(* IEC 61131-3 sources: CODESYS-IO-Visualization/CODESYS-IO-Visualization.fbsproj/Subs/Instruments, 10 files *)

(* ---- Accum.prg.st ---- *)
PROGRAM Accum

VAR_IN_OUT
	Data: Accum_UDT;
END_VAR

VAR
END_VAR

CycleTime(value := Data.CT);
Data.SampleSeconds := Data.SampleSeconds + Data.CT.Sec;

IF (NOT Data.Enable) THEN
	Data.LastEnable := FALSE;
	RETURN;
END_IF;

IF (Data.ValueIn_Realtime < Data.ZeroLimit) THEN
	Data.ValueIn_Realtime := 0.0;
END_IF;

// Set Min / Max Values
IF (Data.ValueIn_Realtime < Data.Value[0].ValueMin) THEN
	Data.Value[0].ValueMin := Data.ValueIn_Realtime;
END_IF;

IF (Data.ValueIn_Realtime > Data.Value[0].ValueMax) THEN
	Data.Value[0].ValueMax := Data.ValueIn_Realtime;
END_IF;

// Check to see if it's time to reset the Total
CASE Data.Period OF
	0: // Manual Reset
		Data.ResetInProcess := Data.Reset OR Data.ResetInternal;
	1: // Hourly
		Data.ResetInProcess := (((Lib_GVL.ClockLocal.Minute = Data.RollMinute) AND (Lib_GVL.ClockLocal.Second < 5)) OR Data.Reset);
	2: // Daily
		Data.ResetInProcess := (((Lib_GVL.ClockLocal.Hour = Data.RollHour) AND (Lib_GVL.ClockLocal.Minute = Data.RollMinute) AND (Lib_GVL.ClockLocal.Second < 5)) OR Data.Reset);
	3: // Monthly
		Data.ResetInProcess := (((Lib_GVL.ClockLocal.Day = Data.RollDay) AND (Lib_GVL.ClockLocal.Hour = Data.RollHour) AND (Lib_GVL.ClockLocal.Minute = Data.RollMinute) AND (Lib_GVL.ClockLocal.Second < 5)) OR Data.Reset);
	4: // Yearly
		Data.ResetInProcess := (((Lib_GVL.ClockLocal.Month = Data.RollMonth) AND (Lib_GVL.ClockLocal.Day = Data.RollDay) AND (Lib_GVL.ClockLocal.Hour = Data.RollHour) AND (Lib_GVL.ClockLocal.Minute = Data.RollMinute) AND (Lib_GVL.ClockLocal.Second < 5)) OR Data.Reset);
END_CASE;

Data.ResetAccumulator := Data.ResetInProcess;

IF (Data.ResetInProcess) THEN	// Always Accum if we are about to reset.
	Data.DoAccum := (Data.SampleSeconds > 0.0);
ELSE  // Only totalize so oftem to limit math errors.  If time change is too big, don't accum this likely means the system clock was updated, just skip it.
	IF (Data.SampleSeconds > (Data.TotalizeInterval * 5)) THEN
		Data.SampleSeconds := 0.0;
	END_IF;
	Data.DoAccum := (Data.SampleSeconds > 0.0) AND (Data.SampleSeconds >= Data.TotalizeInterval) AND (Data.SampleSeconds < (Data.TotalizeInterval * 5));
END_IF;

// Do the Accumulation
IF (Data.DoAccum) THEN
	IF (Data.PauseInternal OR Data.Pause) THEN
		Data.TempAccum := 0.0;
	ELSE
		CASE Data.Mode OF
			0:  // Realtime Value
				Data.TempAccum := Data.ValueIn_Realtime * Data.Gain * (Data.SampleSeconds / Data.Timebase);
			1:  // Reading totalized value that does not reset
				Data.TempAccum := (Data.ValueIn_Total - Data.PrevTotal) * Data.Gain;
			2:  // Reading totalized value that is reset at the device
				Data.TempAccum := Data.ValueIn_Total * Data.Gain;
		ELSE
			Data.TempAccum := 0.0;
		END_CASE;
	END_IF;

	Data.PrevTotal := Data.Value[0].Total;
	Data.SampleSeconds := 0.0;
	Data.Value[0].EndTime := Lib_GVL.ClockLocal;

	CASE Data.Mode OF
		0, 1:  // Realtime Value or Totalized value that does not reset
			IF (ABS(Data.TempAccum) < Data.MaxTotalChange) THEN
				Data.Value[0].Total := Data.Value[0].Total + Data.TempAccum;
			END_IF;
		2:  // Reading totalized value that is reset at the device
			Data.Value[0].Total := Data.TempAccum;
	END_CASE;
END_IF;

// Target Met
Data.TargetMet := (Data.Value[0].Total >= Data.Target);

// Reset the Accumulator
IF (Data.ResetInProcess AND (NOT Data.ResetComplete)) THEN
	FOR Data.i := 8 TO 0 BY -1 DO
		Data.Value[Data.i + 1] := Data.Value[Data.i];
	END_FOR;

	Data.Value[0].ValueMin := Data.ValueIn_Realtime;
	Data.Value[0].ValueMax := Data.ValueIn_Realtime;
	Data.Value[0].Total := 0.0;
	Data.Value[0].EndTime := Lib_GVL.ClockLocal;

	Data.ResetTime := Lib_GVL.ClockLocal.PLCTimeString;
	Data.ResetComplete := TRUE;
	Data.Reset := FALSE;
END_IF;

IF (NOT Data.ResetInProcess) THEN
	Data.ResetComplete := FALSE;
END_IF

(* ---- InstA.prg.st ---- *)
PROGRAM InstA

VAR_IN_OUT
	Data: InstA_UDT;
END_VAR

VAR
END_VAR

// Enable Persist Storage
IF (Data.PersistSize = 0) THEN
	Data.PersistSize := SIZEOF(InstA_UDT);
END_IF;

// Run Value Timer to record 1 second data into a buffer
Data.ValueTimer.In := (NOT Data.ValueTimer.Q);
Timer(TimerData := Data.ValueTimer);

// Handle Manual
CASE Data.Mode OF
	0:	// Online Mode
		Data.TempVal := Data.RawVal;
		Data.CurVal.ClampActive := FALSE;

		IF (Data.CurVal.ClampLowEnable AND (Data.RawVal <= Data.CurVal.ClampLow)) THEN
			Data.TempVal := Data.CurVal.LowRange;
			Data.CurVal.ClampActive := TRUE;
		END_IF;

		IF (Data.CurVal.ClampHighEnable AND (Data.RawVal >= Data.CurVal.ClampHigh)) THEN
			Data.TempVal := Data.CurVal.HighRange;
			Data.CurVal.ClampActive := TRUE;
		END_IF;

		Data.ManualValue := Data.RawVal;

		Data.StatusCode := Data.RawValStatusCode;

		IF (Data.CurVal.ClampActive) THEN
			Data.StatusCode := 129;
		END_IF;

ELSE	// Manual Mode
	Data.TempVal := Data.ManualValue;
	Data.StatusCode := 253;
END_CASE;

// Record the 1 second data into the Value Buffer
IF (Data.ValueCount < 0) THEN
	Data.ValueCount := 0;
END_IF;

IF (Data.ValueTimer.Q) THEN
	Data.ValueCount := Data.ValueCount + 1;
	IF (Data.ValueCount >= 60) THEN
		Data.ValueCount := 60;
	END_IF;

	IF (Data.ValueCount > 1) THEN
		FOR Data.i := (Data.ValueCount - 2) TO 0 BY -1 DO
			Data.ValueBuffer[Data.i + 1] := Data.ValueBuffer[Data.i];
		END_FOR;
		Data.ValueBuffer[0] := Data.TempVal;
	ELSE
		Data.ValueBuffer[0] := Data.TempVal;
	END_IF;
END_IF;

// Set the Avg Value
IF (Data.ValueCount > 1) THEN
	IF (Data.TempVal < Data.CurVal.ValueMin) THEN
		Data.CurVal.ValueMin := Data.TempVal;
	END_IF;

	IF (Data.TempVal > Data.CurVal.ValueMax) THEN
		Data.CurVal.ValueMax := Data.TempVal;
	END_IF;

	Data.ValueSum := 0.0;
	FOR Data.i := 0 TO (Data.ValueCount - 1) DO
		Data.ValueSum := Data.ValueSum + Data.ValueBuffer[Data.i];
	END_FOR;

	// Set the ValueStatus - 0 = Stale, 1 = Decreasing, 2 = Increasing
	Data.CurVal.ValueStatusDly.In := NOT Data.CurVal.ValueStatusDly.Q;
	Timer(TimerData := Data.CurVal.ValueStatusDly);

	IF (Data.CurVal.ValueStatusDly.Q) THEN
		Data.CurVal.ValueAvgPrev := Data.CurVal.ValueAvg;
		IF (Data.ValueBuffer[0] > Data.ValueBuffer[Data.ValueCount - 1]) THEN
			Data.CurVal.ValueStatus := 2;
		END_IF;
		IF (Data.ValueBuffer[0] < Data.ValueBuffer[Data.ValueCount - 1]) THEN
			Data.CurVal.ValueStatus := 1;
		END_IF;
	END_IF;

	// Set the current Average Value
	Data.CurVal.ValueAvg := Data.ValueSum / Data.ValueCount;

// 	IF (Data.CurVal.ValueAvg > Data.CurVal.ValueAvgPrev) THEN
// 		Data.CurVal.ValueStatus := 2;
// 	END_IF;
// 	IF (Data.CurVal.ValueAvg < Data.CurVal.ValueAvgPrev) THEN
// 		Data.CurVal.ValueStatus := 1;
// 	END_IF;
ELSE
	Data.CurVal.ValueAvg := Data.TempVal;
	Data.CurVal.ValueAvgPrev := Data.TempVal;
	Data.CurVal.ValueStatus := 0;
END_IF;

// Set the Percent Value
IF (Data.CurVal.HighRange - Data.CurVal.LowRange) > 0.0 THEN
	Data.CurVal.ValuePct := (Data.CurVal.Value - Data.CurVal.ClampLow) / (Data.CurVal.HighRange - Data.CurVal.LowRange);
ELSE
	Data.CurVal.ValuePct := 0.0;
END_IF

// Reset the Min and Max Values
IF (Data.CurVal.Reset) THEN
	Data.CurVal.ValueMin := Data.TempVal;
	Data.CurVal.ValueMax := Data.TempVal;
	Data.CurVal.Reset := FALSE;
END_IF;

// Set the output values with scaling
IF (Data.DeviceFail.Active) THEN
	CASE Data.FailAction OF
		0: Data.CurVal.Value := Data.FailValue;
		1: Data.CurVal.Value := Data.CurVal.Value;
	ELSE
		Data.CurVal.Value := Data.TempVal;
	END_CASE;
ELSE
	Data.CurVal.Value := Data.TempVal;
END_IF;

// CurVal2 Calculation
InstA_SecondaryValue(Value := Data.CurVal.Value, Data := Data.CurVal2);

// CurVal3 Calculation
InstA_SecondaryValue(Value := Data.CurVal.Value, Data := Data.CurVal3);

// Stale Value
IF (Data.Stale.Enable) THEN
	Data.Stale.StaleTimer.In := (Data.CurVal.Value = Data.Stale.PrevValue);
	Timer(TimerData := Data.Stale.StaleTimer);
	Data.Stale.Detected := Data.Stale.StaleTimer.Q;
	Data.Stale.PrevValue := Data.CurVal.Value;
ELSE
	Data.Stale.Detected := FALSE;
END_IF;

IF (Data.Stale.Detected) THEN
	Data.CurVal.ValueStatus := 0;
	Data.StatusCode := 130;
END_IF;

// Set GlobalStatusCode and String
CASE Data.StatusCode OF
	128: Data.GlobalStatusString := "OK";
	129: Data.GlobalStatusString := "Clamp Active";
	130: Data.GlobalStatusString := "Stale Value";
	253: Data.GlobalStatusString := "Manual Mode";
ELSE
	IF (Data.StatusCode < 128) OR ((Data.StatusCode > 128) AND (Data.StatusCode < 256)) THEN
		Data.GlobalStatusString := "Warning";
	END_IF;

	IF (Data.StatusCode > 255) THEN
		Data.GlobalStatusString := "Failed";
	END_IF;
END_CASE;

Data.GlobalStatusCode := Data.StatusCode + 65536;

AlarmDigital(alarm := Data.OOS);

// Set the input to the Alarms
Data.HiHi.Value := Data.CurVal.Value;
Data.HiHi.OOS := data.OOS.Active;

Data.Hi.Value := Data.CurVal.Value;
Data.Hi.OOS := data.OOS.Active;

Data.Mid2.Value := Data.CurVal.Value;
Data.Mid2.OOS := data.OOS.Active;

Data.Mid1.Value := Data.CurVal.Value;
Data.Mid1.OOS := data.OOS.Active;

Data.Lo.Value := Data.CurVal.Value;
Data.Lo.OOS := data.OOS.Active;

Data.LoLo.Value := Data.CurVal.Value;
Data.LoLo.OOS := data.OOS.Active;

Data.SpDeviation.Value := ABS(Data.HMISP - Data.CurVal.Value);
Data.SpDeviation.OOS := data.OOS.Active;

Data.DeviceFail.OOS := Data.OOS.Active;

Data.DeviceWarning.OOS := Data.OOS.Active;

// Set the Alarm Display Names
Data.DeviceFail.DisplayName := "Fail";
Data.DeviceWarning.DisplayName := "Warning";
Data.HiHi.DisplayName := "HiHi";
Data.Hi.DisplayName := "Hi";
Data.Mid2.DisplayName := "Mid2";
Data.Mid1.DisplayName := "Mid1";
Data.Lo.DisplayName := "Lo";
Data.LoLo.DisplayName := "LoLo";
Data.SpDeviation.DisplayName := "SPDev";

// Run the Alarms
Data.DeviceFail.Value := (Data.StatusCode > 255);
Data.DeviceWarning.Value := (Data.StatusCode > 129);

AlarmDigital(alarm := Data.DeviceFail);
AlarmDigital(alarm := Data.DeviceWarning);

AlarmAnalog(alarm := Data.HiHi);
AlarmAnalog(alarm := Data.Hi);
AlarmAnalog(alarm := Data.Mid2);
AlarmAnalog(alarm := Data.Mid1);
AlarmAnalog(alarm := Data.Lo);
AlarmAnalog(alarm := Data.LoLo);
AlarmAnalog(alarm := Data.SpDeviation);

// Set MaxSeverity and AlarmLevel
Data.MaxSeverity := MAX(Data.DeviceFail.Severity, MAX(Data.DeviceWarning.Severity, MAX(Data.HiHi.Severity, MAX(Data.Hi.Severity, MAX(Data.Mid2.Severity, MAX(Data.Mid1.Severity, MAX(Data.Lo.Severity, MAX(Data.LoLo.Severity, Data.SpDeviation.Severity))))))));

IF (Data.DeviceFail.AlarmLevel + Data.DeviceWarning.AlarmLevel + Data.HiHi.AlarmLevel + Data.Hi.AlarmLevel + Data.Mid2.AlarmLevel + Data.Mid1.AlarmLevel + Data.Lo.AlarmLevel + Data.LoLo.AlarmLevel + Data.SpDeviation.AlarmLevel) > 0 THEN
	Data.AlarmLevel := 6;

	IF (Data.DeviceFail.AlarmLevel > 0) AND (Data.DeviceFail.AlarmLevel < Data.AlarmLevel) THEN
		Data.AlarmLevel := Data.DeviceFail.AlarmLevel;
	END_IF;

	IF (Data.DeviceWarning.AlarmLevel > 0) AND (Data.DeviceWarning.AlarmLevel < Data.AlarmLevel) THEN
		Data.AlarmLevel := Data.DeviceWarning.AlarmLevel;
	END_IF;

	IF (Data.HiHi.AlarmLevel > 0) AND (Data.HiHi.AlarmLevel < Data.AlarmLevel) THEN
		Data.AlarmLevel := Data.HiHi.AlarmLevel;
	END_IF;

	IF (Data.Hi.AlarmLevel > 0) AND (Data.Hi.AlarmLevel < Data.AlarmLevel) THEN
		Data.AlarmLevel := Data.Hi.AlarmLevel;
	END_IF;

	IF (Data.Mid2.AlarmLevel > 0) AND (Data.Mid2.AlarmLevel < Data.AlarmLevel) THEN
		Data.AlarmLevel := Data.Mid2.AlarmLevel;
	END_IF;

	IF (Data.Mid1.AlarmLevel > 0) AND (Data.Mid1.AlarmLevel < Data.AlarmLevel) THEN
		Data.AlarmLevel := Data.Mid1.AlarmLevel;
	END_IF;

	IF (Data.Lo.AlarmLevel > 0) AND (Data.Lo.AlarmLevel < Data.AlarmLevel) THEN
		Data.AlarmLevel := Data.Lo.AlarmLevel;
	END_IF;

	IF (Data.LoLo.AlarmLevel > 0) AND (Data.LoLo.AlarmLevel < Data.AlarmLevel) THEN
		Data.AlarmLevel := Data.LoLo.AlarmLevel;
	END_IF;

	IF (Data.SpDeviation.AlarmLevel > 0) AND (Data.SpDeviation.AlarmLevel < Data.AlarmLevel) THEN
		Data.AlarmLevel := Data.SpDeviation.AlarmLevel;
	END_IF;
ELSE
	Data.AlarmLevel := 0;
END_IF;

// Accumulators
Data.Accum_InUse := FALSE;
FOR Data.i := 0 TO 4 DO
	Data.Accum[Data.i].ValueIn_Realtime := Data.CurVal.Value;
	Data.Accum[Data.i].EU_Realtime := Data.CurVal.EU;
	Data.Accum[Data.i].ValueIn_Total := Data.RawVal_Total;
	Data.Accum[Data.i].PauseInternal := (Data.DeviceFail.Active);
	Accum(Data := Data.Accum[Data.i]);

	IF (Data.Accum[Data.i].Enable) THEN
		Data.Accum_InUse := TRUE;
	END_IF;
END_FOR;

(* ---- InstA_PowerMeter.prg.st ---- *)
PROGRAM InstA_PowerMeter

VAR_IN_OUT
	Data: InstPowerMeter_UDT;
END_VAR

InstA(Data := Data);

InstA(Data := Data.Vab);
InstA(Data := Data.Vbc);
InstA(Data := Data.Vca);
InstA(Data := Data.Vll);
InstA(Data := Data.Van);
InstA(Data := Data.Vbn);
InstA(Data := Data.Vcn);
InstA(Data := Data.Vln);

InstA(Data := Data.Ia);
InstA(Data := Data.Ib);
InstA(Data := Data.Ic);

InstA(Data := Data.kWa);
InstA(Data := Data.kWb);
InstA(Data := Data.kWc);
InstA(Data := Data.kW);

InstA(Data := Data.kVAa);
InstA(Data := Data.kVAb);
InstA(Data := Data.kVAc);
InstA(Data := Data.kVA);

InstA(Data := Data.kVARa);
InstA(Data := Data.kVARb);
InstA(Data := Data.kVARc);
InstA(Data := Data.kVAR);

InstA(Data := Data.PFa);
InstA(Data := Data.PFb);
InstA(Data := Data.PFc);

(* ---- InstA_ROC.prg.st ---- *)
PROGRAM InstA_ROC

VAR_IN_OUT
	Data: InstA_ROC_UDT;
END_VAR

// Enable Persist Storage
IF (Data.PersistSize = 0) THEN
	Data.PersistSize := SIZEOF(InstA_ROC_UDT);
END_IF;

InstA(Data := Data);

(* Rate Of Change Calculations *)
IF (Data.ROCSampleNum < 1) THEN
	Data.ROCSampleNum := 1;
END_IF;

IF (Data.ROCSampleNum > 60) THEN
	Data.ROCSampleNum := 60;
END_IF;

IF (Data.ROCCount < 0) THEN
	Data.ROCCount := 0;
END_IF;

IF (Data.ROCCount > 60) THEN
	Data.ROCCount := 60;
END_IF;

(* Reset the rate of change - Value count > 1 means this block as been running for at least 2 seconds and should have good data *)
IF (Data.ValueCount > 1) THEN
	IF (Data.ROCReset) THEN
		Data.ROCReset := FALSE;
		FOR Data.j := 1 TO 60 BY 1 DO
			Data.ROCBuffer[Data.j] := Data.CurVal.Value;
		END_FOR;
	END_IF;
END_IF;

(* Run ROC Timer *)
Data.ROCTimer.PT := Data.ROCSampleTime;
Data.ROCTimer.In := (NOT Data.ROCTimer.Q);
Timer(TimerData := Data.ROCTimer);

IF (Data.ROCTimer.Q) THEN
	Data.ROCCount := Data.ROCCount + 1;
	IF (Data.ROCCount >= 60) THEN
		Data.ROCCount := 60;
	END_IF;

	IF (Data.ROCCount > 2) THEN
		Data.k := Data.ROCCount - 1;
		WHILE Data.k >= 1 DO
			Data.l := Data.k + 1;
			Data.ROCBuffer[Data.l] := Data.ROCBuffer[Data.k];
			Data.k := Data.k - 1;
		END_WHILE;
		Data.ROCBuffer[1] := Data.CurVal.Value;
	ELSE
		Data.ROCBuffer[1] := Data.CurVal.Value;
	END_IF;
END_IF;

IF (Data.ValueCount > 1) AND (NOT Data.OOS.Active) THEN
	Data.CurValROC := Data.CurVal.Value - Data.ROCBuffer[Data.ROCSampleNum - 1];
ELSE
	Data.CurValROC := 0.0;
END_IF;

CASE Data.CurValROC2_Mode OF
	1: // (m * x) + b
		Data.CurValROC2 := (Data.CurValROC * Data.CurValROC2_Mult) + Data.CurValROC2_Offset;

	2: // (m * x) + b
		Data.CurValROC2 := (Data.CurValROC + Data.CurValROC2_Offset) * Data.CurValROC2_Mult;
END_CASE;

Data.ROCHi.Value := Data.CurValROC;
Data.ROCLo.Value := Data.CurValROC;

AlarmAnalog(alarm := Data.ROCHi);
AlarmAnalog(alarm := Data.ROCLo);

(* ---- InstA_SecondaryValue.prg.st ---- *)
PROGRAM InstA_SecondaryValue

VAR_INPUT
	Value: REAL;
END_VAR

VAR_IN_OUT
	Data: InstA_Value_Settings2_UDT;
END_VAR

CASE Data.Mode OF
	1: // (m * x) + b
		Data.Value := (Value * Data.Multiplier) + Data.Offset;

	2: // (m * x) + b
		Data.Value := (Value + Data.Offset) * Data.Multiplier;
END_CASE;

(* ---- InstA_SetAccumMode.prg.st ---- *)
PROGRAM InstA_SetAccumMode

VAR_IN_OUT
	Data: InstA_UDT;	// The InstA_UDT to Modify
END_VAR

VAR_INPUT
	Mode: INT;	// 0 = Realtime Totalizer, 1 = Read Meter Total (No Reset), 2 = Read Meter Total (with Reset)
END_VAR

VAR
	i: INT;
END_VAR

// Set Accumulator Mode
// 0 = Realtime Totalizer, 1 = Read Meter Total (No Reset), 2 = Read Meter Total (with Reset)

IF (Mode < 0) THEN
	Mode := 0;
END_IF;

IF (Mode > 2) THEN
	Mode := 2;
END_IF;

FOR i := 0 TO 4 DO
	Data.Accum[i].Mode := Mode;
END_FOR;

(* ---- InstD.prg.st ---- *)
PROGRAM InstD

VAR_IN_OUT
	Data: InstD_UDT;
END_VAR

VAR
END_VAR

// Enable Persist Storage
IF (Data.PersistSize = 0) THEN
	Data.PersistSize := SIZEOF(InstD_UDT);
END_IF;

// Handle Manual
CASE Data.Mode OF
	0:	// Online Mode
		Data.TempVal := Data.RawVal;
		Data.ManualValue := Data.RawVal;
		Data.StatusCode := Data.RawValStatusCode;
ELSE	// Manual Mode
	Data.TempVal := Data.ManualValue;
	Data.StatusCode := 253;
END_CASE;

// Set the output value
IF (Data.DeviceFail.Active) THEN
	CASE Data.FailAction OF
		0: Data.CurVal := Data.FailValue;
		1: Data.CurVal := Data.CurVal;
	ELSE
		Data.CurVal := Data.TempVal;
	END_CASE;
ELSE
	Data.CurVal := Data.TempVal;
END_IF;

// Set GlobalStatusCode and String
CASE Data.StatusCode OF
	128: Data.GlobalStatusString := "OK";
	253: Data.GlobalStatusString := "Manual Mode";
ELSE
	IF (Data.StatusCode < 128) OR ((Data.StatusCode > 128) AND (Data.StatusCode < 256)) THEN
		Data.GlobalStatusString := "Warning";
	END_IF;

	IF (Data.StatusCode > 255) THEN
		Data.GlobalStatusString := "Failed";
	END_IF;
END_CASE;

Data.GlobalStatusCode := Data.StatusCode + 65536;

// Set OOS Inputs
AlarmDigital(alarm := Data.OOS);
Data.DeviceFail.OOS := Data.OOS.Active;
Data.DeviceWarning.OOS := Data.OOS.Active;
Data.Process.OOS := Data.OOS.Active;

// Set the Alarm Display Names
Data.DeviceFail.DisplayName := "Fail";
Data.DeviceWarning.DisplayName := "Warning";
Data.Process.DisplayName := "Process";

// Run the Alarms
Data.DeviceFail.Value := (Data.StatusCode > 255);
Data.DeviceWarning.Value := (Data.StatusCode > 128);
Data.Process.Value := Data.CurVal;

AlarmDigital(alarm := Data.DeviceFail);
AlarmDigital(alarm := Data.DeviceWarning);
AlarmDigital(alarm := Data.Process);

Data.MaxSeverity := MAX(Data.DeviceFail.Severity, MAX(Data.DeviceWarning.Severity, Data.Process.Severity));

IF (Data.DeviceFail.AlarmLevel + Data.DeviceWarning.AlarmLevel + Data.Process.AlarmLevel) > 0 THEN
	Data.AlarmLevel := 6;

	IF (Data.DeviceFail.AlarmLevel > 0) AND (Data.DeviceFail.AlarmLevel < Data.AlarmLevel) THEN
		Data.AlarmLevel := Data.DeviceFail.AlarmLevel;
	END_IF;

	IF (Data.DeviceWarning.AlarmLevel > 0) AND (Data.DeviceWarning.AlarmLevel < Data.AlarmLevel) THEN
		Data.AlarmLevel := Data.DeviceWarning.AlarmLevel;
	END_IF;

	IF (Data.Process.AlarmLevel > 0) AND (Data.Process.AlarmLevel < Data.AlarmLevel) THEN
		Data.AlarmLevel := Data.Process.AlarmLevel;
	END_IF;
ELSE
	Data.AlarmLevel := 0;
END_IF;

(* ---- MapInstAFromIO.prg.st ---- *)
PROGRAM MapInstAFromIO

VAR_IN_OUT
	Data: InstA_UDT;
	IO: Channel_UDT;
END_VAR

Data.RawVal := IO.ValueEu;
Data.RawValStatusCode := IO.StatusCode + 128;

// Map Simulation Settings to IO
IO.SimulationEnable := (NOT Data.Sim.SimDisable);
IO.Simulator.irChangeRate := Data.Sim.ChangeRate;
IO.Simulator.irNoisePct := Data.Sim.NoisePct;
IO.Simulator.irHighLimit := Data.CurVal.HighRange;
IO.Simulator.irLowLimit := Data.CurVal.LowRange;
IO.Simulator.odiStatusCode := Data.Sim.StatusCode;

IF (Data.CurVal.HighRange - Data.CurVal.LowRange) > 0 THEN
	IO.Simulator.irPercent := (Data.Sim.RawVal / (Data.CurVal.HighRange - Data.CurVal.LowRange)) * 100.0;
ELSE
	IO.Simulator.irPercent := Data.Sim.RawVal;
END_IF;

(* ---- MapInstAFromValue.prg.st ---- *)
PROGRAM MapInstAFromValue
VAR_IN_OUT
	Data: InstA_UDT;
END_VAR

VAR_INPUT
	Value: REAL;
	Status: DINT;
	Total: REAL := 0.0;
END_VAR

VAR
	i: INT;
END_VAR

Data.RawVal := Value;

IF Status < 0 THEN
	Data.RawValStatusCode := -1;
ELSE
	Data.RawVal := Value;
	Data.RawValStatusCode := Status;
END_IF;

// Accumulators
FOR i := 0 TO 4 DO
	Data.Accum[i].ValueIn_Total := Total;
END_FOR;

(* ---- MapInstDFromIO.prg.st ---- *)
PROGRAM MapInstDFromIO
VAR_IN_OUT
	Data: InstD_UDT;
	IO: Channel_UDT;
END_VAR

Data.RawVal := IO.ValueDig;
Data.RawValStatusCode := IO.StatusCode + 128;

// Map Simulation Settings to IO
IO.SimulationEnable := (NOT Data.Sim.SimDisable);
IO.Simulator.ibValue := Data.Sim.RawVal;
IO.Simulator.odiStatusCode := Data.Sim.StatusCode;
